// TIA Portal project "Profikum" (V17)

(* hardware
DEVICE "S7-1500/ET200MP-Station_1"  S7-1500 station
   slot 0: "Profilschiene_0"  Rack  6ES7 590-1***0-0AA0
   slot 1: "workstation2.cpu"  CPU 1516-3 PN/DP  6ES7 516-3AN01-0AB0  V2.9
      slot 3: "CPU-Display_1"  6ES7591-1BA00-0AA0
      slot 32768: "PROFINET-Schnittstelle_1"  X1
      slot 33024: "PROFINET-Schnittstelle_2"  X2
      slot 33280: "DP-Schnittstelle_1"  X3
      slot 34817: "Virtual CP interface port_1"  Virtual CP interface port  Virtual CP interface port
DEVICE "S7-1500/ET200MP-Station_2"  S7-1500 station
   slot 0: "Profilschiene_0"  Rack  6ES7 590-1***0-0AA0
   slot 1: "workstation2.rio"  IM 155-5 PN ST  6ES7 155-5AA00-0AB0  V3.0
   slot 2: "DI 32x24VDC HF_1"  DI 32x24VDC HF  6ES7 521-1BL00-0AB0  V2.0
   slot 3: "DQ 32x24VDC/0.5A HF_1"  DQ 32x24VDC/0.5A HF  6ES7 522-1BL01-0AB0  V1.0
   slot 4: "AI 8xU/I/RTD/TC ST_1"  AI 8xU/I/RTD/TC ST  6ES7 531-7KF00-0AB0  V2.0
   slot 5: "AQ 8xU/I HS_1"  AQ 8xU/I HS  6ES7 532-5HF00-0AB0  V2.0
DEVICE "GSD-Geraet_1"  GSD.Device.PN
   slot 0: "Baugruppenträger"  Rack  V1.0
   slot 0: "workstation2.profikum"  Profikum  123 444 555  V0.1.1
      slot 0: "Profikum"  Profikum
      slot 1: "X1"  X1
         slot 1: "X1 P1"  X1 P1
      slot 1: "Motors_1"  Motors  1.0
         slot 0: "Motors submodule"  Motors submodule
   slot 2: "IMU sensors_1"  IMU sensors  1.0
      slot 0: "Acceleration"  Acceleration
      slot 1: "Gyro"  Gyro
      slot 2: "Magnetometer"  Magnetometer
   slot 3: "Ultrasound distance sensor_1"  Ultrasound distance sensor  1.0
      slot 0: "Ultrasound distance sensor"  Ultrasound distance sensor
   slot 4: "Encoder_1"  Encoder  1.0
      slot 0: "Motor Encoder"  Motor Encoder
   slot 5: "Debug_1"  Debug  1.0
      slot 0: "Debug"  Debug
*)

// ===== PLC "workstation2.cpu"  CPU 1516-3 PN/DP =====

VAR_GLOBAL   // PLC tag table "Standard-Variablentabelle"
   "profikumOutputs" AT %I100.0 : "typeProfikumOutputs";
   "profikumInputs" AT %Q100.0 : "typeProfikumInputs";
   "leftButton" AT %I0.0 : Bool;
   "rightButton" AT %I0.1 : Bool;
   "autoModeButton" AT %I0.2 : Bool;
END_VAR

TYPE "typeProfikumOutputs"
VERSION : 0.1
   STRUCT
      accelerationX : Int;
      accelerationY : Int;
      accelerationZ : Int;
      gyroX : Int;
      gyroY : Int;
      gyroZ : Int;
      magnetometerX : Int;
      magnetometerY : Int;
      magnetometerZ : Int;
      distanceRight_mm : Int;
      distanceLeft_mm : Int;
      leftDistance_mm : Int;
      rightDistance_mm : Int;
      leftSpeed_mm_s : Int;
      rightSpeed_mm_s : Int;
      scalingLeft : Int;
      scalingRight : Int;
      scalingDiff : Int;
   END_STRUCT;
END_TYPE

TYPE "typeProfikumInputs"
VERSION : 0.1
   STRUCT
      leftMotorSpeed : Int;
      rightMotorSpeed : Int;
   END_STRUCT;
END_TYPE

TYPE "typeProfikumParameters"
   STRUCT
      v : LReal := 0.3;   // m/s
      DeltaYCont : LReal := 0.2;   // Distance, which corresponds via Tcont=DeltaYCont/v to the time constant of the controller
      relTobs : LReal := 0.5;   // Tobs=relTobs*Tcont
      d : LReal := 0.09;   // meters. Distance between the wheels
      vStand : LReal := 0.03;   // m/s. Speed, under which we assume the stand-still model for the observer
      TobsStand : LReal := 1.0;   // s. Time constant observer of the stand-still model.
      phiMax : LReal := 0.175;   // rad. Maximal angle we want to allow. 0.175rad=10°
      uMax : LReal := 0.78525;   // Maximal input we want to allow. 0.78525 rad/s = 45°/s
      scaleU : LReal := 1.0;
   END_STRUCT;
END_TYPE

TYPE "typeProfikumController"
   STRUCT
      phi : LReal;   // Angle of the robot, relative to the wall, in rad
      x : LReal := 0.25;   // Estimated distance robot from wall, in meters
      w : LReal := 0.25;   // Set distance robot from wall, in meters
      p : "typeProfikumParameters";   // Parameters of the bot
   END_STRUCT;
END_TYPE

DATA_BLOCK "InstManualControl"   // DB1
{ S7_Optimized_Access := 'TRUE' }
VERSION : 0.1
// stored: InstanceOfName ManualControl
"ManualControl"
BEGIN
END_DATA_BLOCK

DATA_BLOCK "InstCurveControl"   // DB2
{ S7_Optimized_Access := 'TRUE' }
VERSION : 0.1
// stored: InstanceOfName CurveControl
"CurveControl"
BEGIN
END_DATA_BLOCK

DATA_BLOCK "ProfikumController"   // DB3
{ S7_Optimized_Access := 'TRUE' }
VERSION : 0.1
BEGIN
END_DATA_BLOCK

DATA_BLOCK "VisualizationVars"   // DB4
{ S7_Optimized_Access := 'TRUE' }
VERSION : 0.1
   VAR
      xMeas : LReal;
      x : LReal;
      phi : LReal;
      u : LReal;
      uMeas : LReal;
      vLeft : LReal;
      vRight : LReal;
      v : LReal;
      vLeftMeas : LReal;
      vRightMeas : LReal;
      vMeas : LReal;
   END_VAR
BEGIN
END_DATA_BLOCK

FUNCTION_BLOCK "ManualControl"   // FB1, SCL
{ S7_Optimized_Access := 'TRUE' }
VERSION : 0.1
   VAR_INPUT
      leftButtonPressed : Bool;
      rightButtonPressed : Bool;
      vOn : LReal;
   END_VAR
   VAR_OUTPUT
      leftSpeed : LReal;
      rightSpeed : LReal;
   END_VAR
BEGIN
   IF #leftButtonPressed THEN
       #leftSpeed := #vOn;
   ELSE
       #leftSpeed := 0;
   END_IF;

   IF #rightButtonPressed THEN
       #rightSpeed := #vOn;
   ELSE
       #rightSpeed := 0;
   END_IF;
END_FUNCTION_BLOCK

FUNCTION_BLOCK "CurveControl"   // FB2, SCL
{ S7_Optimized_Access := 'TRUE' }
VERSION : 0.1
   VAR_INPUT
      leftButtonPressed : Bool;
      rightButtonPressed : Bool;
      vOn : LReal;
   END_VAR
   VAR_OUTPUT
      leftSpeed : LReal;
      rightSpeed : LReal;
   END_VAR
   VAR_TEMP
      t : LReal;
   END_VAR
   VAR CONSTANT
      PI : LReal := 3.1415927;
   END_VAR
BEGIN
   #t := LINT_TO_LREAL(TIME_TO_LINT(TIME_TCK())) / 1000.0;
   IF #leftButtonPressed THEN
       #leftSpeed := #vOn * (0.9+0.4*SIN(2 * #PI * #t /4.0));
       #rightSpeed := #vOn * (0.9+0.4*SIN(2 * #PI * #t / 4.0+#PI/2));
   ELSIF #rightButtonPressed THEN
       #leftSpeed :=#vOn;
       #rightSpeed := #vOn;
   ELSE
       #leftSpeed := 0; 
       #rightSpeed := 0;
   END_IF;
END_FUNCTION_BLOCK

FUNCTION "ProfikumMotor" : Void   // FC1, SCL
{ S7_Optimized_Access := 'TRUE' }
VERSION : 0.1
   VAR_INPUT
      leftSpeed : LReal;   // in m/s.
      rightSpeed : LReal;   // in m/s.
   END_VAR
   VAR_OUTPUT
      leftSpeedRaw : Int;
      rightSpeedRaw : Int;
   END_VAR
BEGIN
   #leftSpeedRaw := LREAL_TO_INT(#leftSpeed * 1000);
   #rightSpeedRaw := LREAL_TO_INT(#rightSpeed *1000);
END_FUNCTION

FUNCTION "Observer" : Void   // FC2, SCL
{ S7_Optimized_Access := 'TRUE' }
VERSION : 0.1
   VAR_INPUT
      phi : LReal;
      y : LReal;
      u : LReal;
      p : "typeProfikumParameters";
      yMeasured : LReal;
   END_VAR
   VAR_OUTPUT
      dphi : LReal;
      dy : LReal;
   END_VAR
   VAR_TEMP
      p1 : LReal;
      p2 : LReal;
      v : LReal;
      "e" : LReal;
   END_VAR
BEGIN
   // Calculate parameters of observer
   #v := #p.v;
   #p1 := 1.0 / #v / #p.DeltaYCont**2;
   #p2 := 2.0 / #p.DeltaYCont;

   // Calculate error
   #e := #yMeasured - #y;

   // Calculate derivatives
   #dphi := 2.0 * #v / #p.d * #u + #p1 * #e;
   #dy := #v * #phi + #p2 * #e;
END_FUNCTION

ORGANIZATION_BLOCK "Main"   // OB1, LAD, ProgramCycle
TITLE = "Main Program Sweep (Cycle)"
{ S7_Optimized_Access := 'TRUE' }
VERSION : 0.1
   VAR_INPUT
      Initial_Call : Bool;   // Initial call of this OB
      Remanence : Bool;   // =True, if remanent data are available
   END_VAR
   VAR_TEMP
      tempLeftSpeed : LReal;
      tempRightSpeed : LReal;
   END_VAR
   VAR_TEMP   // added for the SCL form of the ladder/FBD networks
      _w1 : Bool;
   END_VAR
BEGIN

REGION Network 1
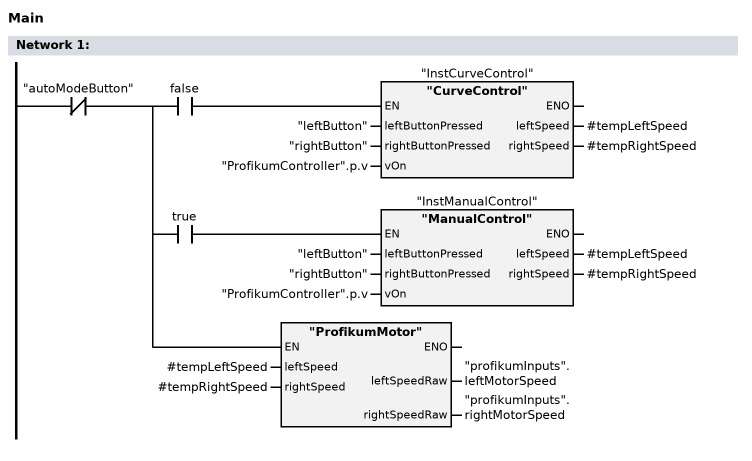
   RUNG wire#powerrail
      I_Contact( "autoModeButton" )
      wire#w1
      Contact( false )
      "InstCurveControl"(leftButtonPressed := "leftButton", rightButtonPressed := "rightButton", vOn := "ProfikumController".p.v, leftSpeed => #tempLeftSpeed, rightSpeed => #tempRightSpeed)
   END_RUNG
   RUNG wire#w1
      Contact( true )
      "InstManualControl"(leftButtonPressed := "leftButton", rightButtonPressed := "rightButton", vOn := "ProfikumController".p.v, leftSpeed => #tempLeftSpeed, rightSpeed => #tempRightSpeed)
   END_RUNG
   RUNG wire#w1
      "ProfikumMotor"(leftSpeed := #tempLeftSpeed, rightSpeed := #tempRightSpeed, leftSpeedRaw => "profikumInputs".leftMotorSpeed, rightSpeedRaw => "profikumInputs".rightMotorSpeed)
   END_RUNG
   // the same network as SCL:
   #_w1 := NOT "autoModeButton";
   IF NOT "autoModeButton" AND false THEN
       "InstCurveControl"(leftButtonPressed := "leftButton",   // "CurveControl"
                          rightButtonPressed := "rightButton",
                          vOn := "ProfikumController".p.v,
                          leftSpeed => #tempLeftSpeed,
                          rightSpeed => #tempRightSpeed);
   END_IF;
   IF #_w1 AND true THEN
       "InstManualControl"(leftButtonPressed := "leftButton",   // "ManualControl"
                           rightButtonPressed := "rightButton",
                           vOn := "ProfikumController".p.v,
                           leftSpeed => #tempLeftSpeed,
                           rightSpeed => #tempRightSpeed);
   END_IF;
   IF #_w1 THEN
       "ProfikumMotor"(leftSpeed := #tempLeftSpeed,
                       rightSpeed := #tempRightSpeed,
                       leftSpeedRaw => "profikumInputs".leftMotorSpeed,
                       rightSpeedRaw => "profikumInputs".rightMotorSpeed);
   END_IF;
END_REGION
END_ORGANIZATION_BLOCK

ORGANIZATION_BLOCK "ControllerMain"   // OB30, SCL, CyclicInterrupt
{ S7_Optimized_Access := 'TRUE' }
VERSION : 0.1
   VAR_INPUT
      Initial_Call : Bool;   // Initial call of this OB
      Event_Count : Int;   // Events discarded
   END_VAR
   VAR_TEMP
      xMeas : LReal;
      p : "typeProfikumParameters";
      v : LReal;
      Tcont : LReal;
      Tobs : LReal;
      k1 : LReal;
      k2 : LReal;
      l1 : LReal;
      l2 : LReal;
      x : LReal;
      phi : LReal;
      w : LReal;
      dx : LReal;
      dphi : LReal;
      u : LReal;
      uMeas : LReal;
      Kpre : LReal;
      vLeft : LReal;
      vRight : LReal;
      Delta_v : LReal;
      vLeftRaw : Int;
      vRightRaw : Int;
      vMeas : LReal;
   END_VAR
   VAR CONSTANT
      PI : LReal := 3.14159265359;
      "dt" : LReal := 0.032;   // Integration time constant in s. Must be the same as the period of the OB.
   END_VAR
BEGIN
   // Copy states etc. into temporary variables for easier access
   #x := "ProfikumController".x;
   #phi := "ProfikumController".phi;
   #w := "ProfikumController".w;
   #p := "ProfikumController".p;
   #v := #p.v;

   // Get measured distance to wall (in m)
   #xMeas := INT_TO_LREAL("profikumOutputs".distanceRight_mm) / 1000.0;
   IF #xMeas <= 0 THEN
       // Assume observer is perfect in case of an invalid measurement
       #xMeas := #x;
   END_IF;
   // Current speed (in m/s) = average left and right speed
   #vMeas := INT_TO_LREAL("profikumOutputs".leftSpeed_mm_s + "profikumOutputs".rightSpeed_mm_s) / 1000.0 / 2.0;
   #uMeas := 1.0 / #p.d * ("profikumOutputs".rightSpeed_mm_s - "profikumOutputs".leftSpeed_mm_s) / 1000.0;

   // Only run controller if speed is nonzero
   IF "autoModeButton" AND ABS(#v) >= #p.vStand THEN
       // Time constant controller and observer
       #Tcont := #p.DeltaYCont / #v;
       #Tobs := #p.relTobs * #Tcont;

       // Parameters controller and observer
       #k1 := 1.0 / ((#Tcont ** 2) * #v);
       #k2 := 2.0 / #Tcont;
       #l1 := + 2.0 / #Tobs;
       #l2 := + 1.0 / ((#Tobs ** 2) * #v);

       // Pre-filter
       #Kpre := 1.0 / (#v * (#Tcont ** 2.0));

       // Controller
       #u := - #k1 * #x - #k2*#phi + #Kpre * #w;
       // Prevent to large angles
       //IF (#u > 0 AND #phi >= #p.phiMax) OR (#u < 0 AND #phi <= - #p.phiMax) THEN
           //#u := 0;
       IF #u > #p.uMax THEN
           #u := #p.uMax;
       ELSIF #u < - #p.uMax THEN
           #u := - #p.uMax;
       END_IF;

       // Observer ODEs
       #dx := SIN(#phi) * #v + #l1 * (#xMeas - #x);
       #dphi := #u + #l2 * (#xMeas - #x);

       // Integrate observer
       #x := #x + #dx * #dt;
       #phi := #phi + #dphi * #dt;


   ELSE
       // Stand still model. We still learn the position, but don't take any control actions nor update our angle estimate.
       #dx := 1.0 / #p.TobsStand * (#xMeas - #x);
       #dphi := 1.0 / #p.TobsStand * -#phi;
       #x := #x + #dx * #dt;
       #phi := #phi + #dphi * #dt;
       #u := 0.0;
   END_IF;

   // Save state of observer
   "ProfikumController".x := #x;
   "ProfikumController".phi := #phi;

   // Calculate speeds of motors
   #Delta_v := #p.d * #u * #p.scaleU;
   #vLeft  := #v - #Delta_v / 2.0;
   #vRight := #v + #Delta_v / 2.0;

   "ProfikumMotor"(leftSpeed := #vLeft,
                   rightSpeed := #vRight,
                   leftSpeedRaw => #vLeftRaw,
                   rightSpeedRaw => #vRightRaw);

   // Only "activate" controller if we are in auto-mode. Otherwise, effectively, only the observer is running.
   IF "autoModeButton" THEN
       "profikumInputs".leftMotorSpeed := #vLeftRaw;
       "profikumInputs".rightMotorSpeed := #vRightRaw;
   END_IF;

   "VisualizationVars".xMeas := #xMeas;
   "VisualizationVars".x := #x;
   "VisualizationVars".phi := #phi/#PI*180;
   "VisualizationVars".u := #u / #PI * 180;
   "VisualizationVars".uMeas := #uMeas / #PI * 180;

   "VisualizationVars".vLeft := #vLeft;
   "VisualizationVars".vRight := #vRight;
   "VisualizationVars".v := (#vLeft+#vRight)/2.0;

   "VisualizationVars".vLeftMeas := INT_TO_LREAL("profikumOutputs".leftSpeed_mm_s) / 1000;
   "VisualizationVars".vRightMeas := INT_TO_LREAL("profikumOutputs".rightSpeed_mm_s) / 1000;
   "VisualizationVars".vMeas := #v;
END_ORGANIZATION_BLOCK